// TIA Portal V20 export
TYPE "UDT_SelSt"
   STRUCT
      b0 : Byte;   // Byte 0
      b1 : Byte;   // Byte 1
      b2 : Byte;   // Byte 2
      b3 : Byte;   // Byte 3
      b4 : Byte;   // Byte 4
      b5 : Byte;   // Byte 5
      b6 : Byte;   // Byte 6
      b7 : Byte;   // Byte 7
      b8 : Byte;   // Byte 8
      b9 : Byte;   // Byte 9
      b10 : Byte;   // Byte 10
      b11 : Byte;   // Byte 11
      b12 : Byte;   // Byte 12
      b13 : Byte;   // Byte 13
      b14 : Byte;   // Byte 14
      b15 : Byte;   // Byte 15
   END_STRUCT;
END_TYPE
